(* Logix 5000 project; controller R1USB70001_CWRU_Scenario_Gen_20111116 vendor 1 type 14 code 54 rev 19.11; software revision 19.01; part 5 of 9 *)
(* tags used below, declared in another part *)
   EditScenarioPv : EditScenarioPv;
   ExecutePv : ExecutePv;
   CalcRemainTimeIndex : DINT;
   CalcTotalTimeIndex : DINT;
   CL_LP_B2_SG : ALIAS FOR ACNR_CP_SG_N5:2:O.4;
   EditScenario : EditScenarioPub;
   Execute : ExecutePub;
   HMI : HMIPub;
   IL_LP_B1_SG : ALIAS FOR ACNR_CP_SG_N5:4:O.1;
   IL_LP_B2_SG : ALIAS FOR ACNR_CP_SG_N5:5:O.4;
   IL_LP_ML_SG : ALIAS FOR ACNR_CP_SG_N5:4:O.0;
   Scenario : Scenario_Def[100];
   TimeTblStepNmbr : DINT;
(* MainProgram, continued *)

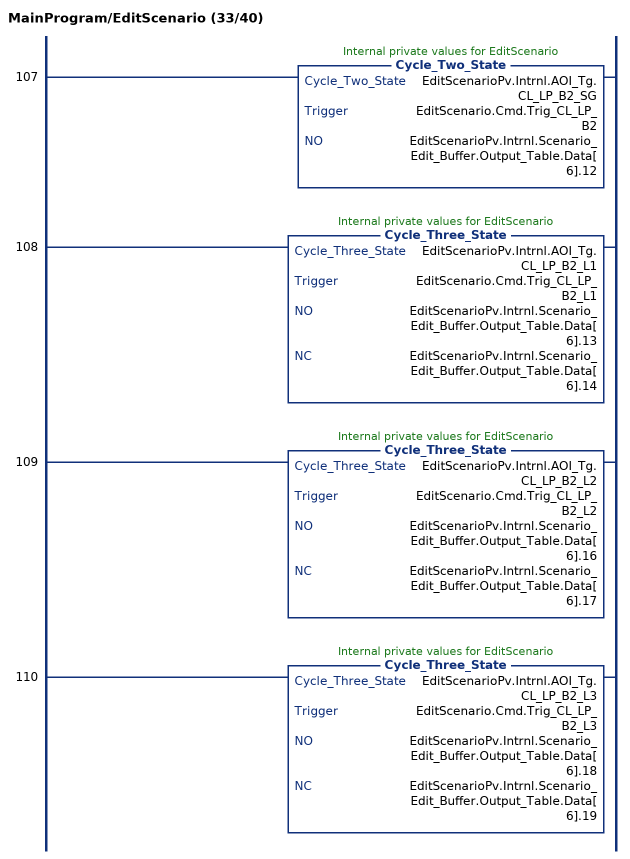
   107: Cycle_Two_State(EditScenarioPv.Intrnl.AOI_Tg.CL_LP_B2_SG,EditScenario.Cmd.Trig_CL_LP_B2,EditScenarioPv.Intrnl.Scenario_Edit_Buffer.Output_Table.Data[6].12);
   108: Cycle_Three_State(EditScenarioPv.Intrnl.AOI_Tg.CL_LP_B2_L1,EditScenario.Cmd.Trig_CL_LP_B2_L1,EditScenarioPv.Intrnl.Scenario_Edit_Buffer.Output_Table.Data[6].13,EditScenarioPv.Intrnl.Scenario_Edit_Buffer.Output_Table.Data[6].14);
   109: Cycle_Three_State(EditScenarioPv.Intrnl.AOI_Tg.CL_LP_B2_L2,EditScenario.Cmd.Trig_CL_LP_B2_L2,EditScenarioPv.Intrnl.Scenario_Edit_Buffer.Output_Table.Data[6].16,EditScenarioPv.Intrnl.Scenario_Edit_Buffer.Output_Table.Data[6].17);
   110: Cycle_Three_State(EditScenarioPv.Intrnl.AOI_Tg.CL_LP_B2_L3,EditScenario.Cmd.Trig_CL_LP_B2_L3,EditScenarioPv.Intrnl.Scenario_Edit_Buffer.Output_Table.Data[6].18,EditScenarioPv.Intrnl.Scenario_Edit_Buffer.Output_Table.Data[6].19);
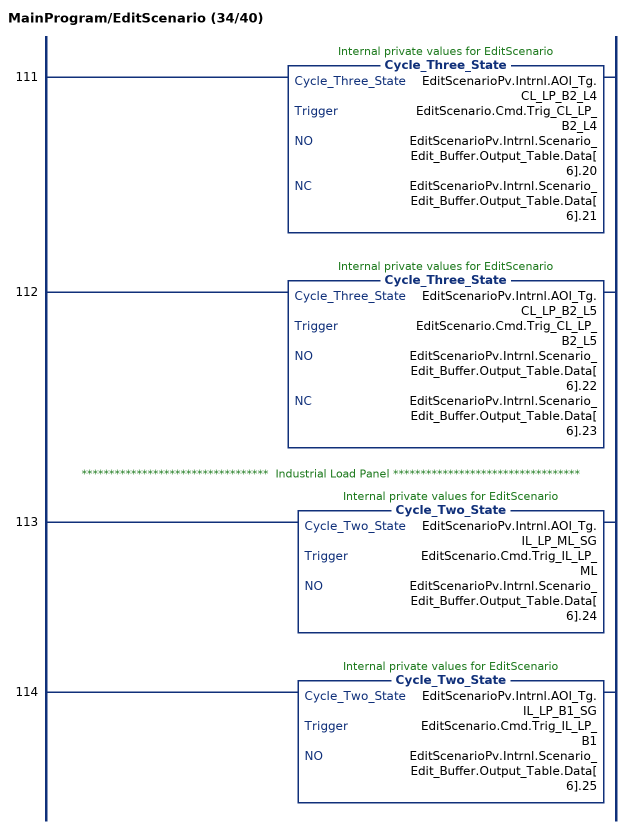
   111: Cycle_Three_State(EditScenarioPv.Intrnl.AOI_Tg.CL_LP_B2_L4,EditScenario.Cmd.Trig_CL_LP_B2_L4,EditScenarioPv.Intrnl.Scenario_Edit_Buffer.Output_Table.Data[6].20,EditScenarioPv.Intrnl.Scenario_Edit_Buffer.Output_Table.Data[6].21);
   112: Cycle_Three_State(EditScenarioPv.Intrnl.AOI_Tg.CL_LP_B2_L5,EditScenario.Cmd.Trig_CL_LP_B2_L5,EditScenarioPv.Intrnl.Scenario_Edit_Buffer.Output_Table.Data[6].22,EditScenarioPv.Intrnl.Scenario_Edit_Buffer.Output_Table.Data[6].23);
   // **********************************  Industrial Load Panel **********************************
   113: Cycle_Two_State(EditScenarioPv.Intrnl.AOI_Tg.IL_LP_ML_SG,EditScenario.Cmd.Trig_IL_LP_ML,EditScenarioPv.Intrnl.Scenario_Edit_Buffer.Output_Table.Data[6].24);
   114: Cycle_Two_State(EditScenarioPv.Intrnl.AOI_Tg.IL_LP_B1_SG,EditScenario.Cmd.Trig_IL_LP_B1,EditScenarioPv.Intrnl.Scenario_Edit_Buffer.Output_Table.Data[6].25);
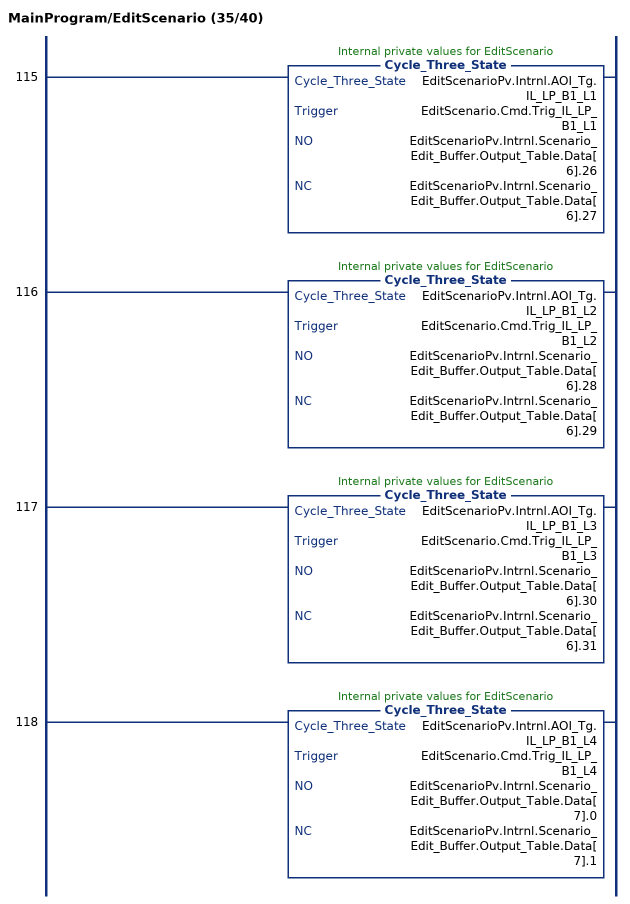
   115: Cycle_Three_State(EditScenarioPv.Intrnl.AOI_Tg.IL_LP_B1_L1,EditScenario.Cmd.Trig_IL_LP_B1_L1,EditScenarioPv.Intrnl.Scenario_Edit_Buffer.Output_Table.Data[6].26,EditScenarioPv.Intrnl.Scenario_Edit_Buffer.Output_Table.Data[6].27);
   116: Cycle_Three_State(EditScenarioPv.Intrnl.AOI_Tg.IL_LP_B1_L2,EditScenario.Cmd.Trig_IL_LP_B1_L2,EditScenarioPv.Intrnl.Scenario_Edit_Buffer.Output_Table.Data[6].28,EditScenarioPv.Intrnl.Scenario_Edit_Buffer.Output_Table.Data[6].29);
   117: Cycle_Three_State(EditScenarioPv.Intrnl.AOI_Tg.IL_LP_B1_L3,EditScenario.Cmd.Trig_IL_LP_B1_L3,EditScenarioPv.Intrnl.Scenario_Edit_Buffer.Output_Table.Data[6].30,EditScenarioPv.Intrnl.Scenario_Edit_Buffer.Output_Table.Data[6].31);
   118: Cycle_Three_State(EditScenarioPv.Intrnl.AOI_Tg.IL_LP_B1_L4,EditScenario.Cmd.Trig_IL_LP_B1_L4,EditScenarioPv.Intrnl.Scenario_Edit_Buffer.Output_Table.Data[7].0,EditScenarioPv.Intrnl.Scenario_Edit_Buffer.Output_Table.Data[7].1);
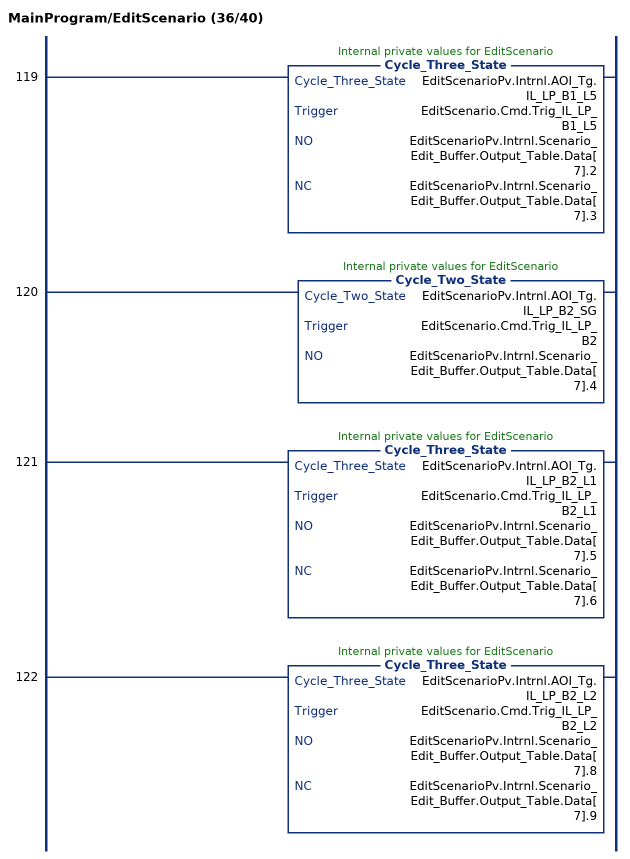
   119: Cycle_Three_State(EditScenarioPv.Intrnl.AOI_Tg.IL_LP_B1_L5,EditScenario.Cmd.Trig_IL_LP_B1_L5,EditScenarioPv.Intrnl.Scenario_Edit_Buffer.Output_Table.Data[7].2,EditScenarioPv.Intrnl.Scenario_Edit_Buffer.Output_Table.Data[7].3);
   120: Cycle_Two_State(EditScenarioPv.Intrnl.AOI_Tg.IL_LP_B2_SG,EditScenario.Cmd.Trig_IL_LP_B2,EditScenarioPv.Intrnl.Scenario_Edit_Buffer.Output_Table.Data[7].4);
   121: Cycle_Three_State(EditScenarioPv.Intrnl.AOI_Tg.IL_LP_B2_L1,EditScenario.Cmd.Trig_IL_LP_B2_L1,EditScenarioPv.Intrnl.Scenario_Edit_Buffer.Output_Table.Data[7].5,EditScenarioPv.Intrnl.Scenario_Edit_Buffer.Output_Table.Data[7].6);
   122: Cycle_Three_State(EditScenarioPv.Intrnl.AOI_Tg.IL_LP_B2_L2,EditScenario.Cmd.Trig_IL_LP_B2_L2,EditScenarioPv.Intrnl.Scenario_Edit_Buffer.Output_Table.Data[7].8,EditScenarioPv.Intrnl.Scenario_Edit_Buffer.Output_Table.Data[7].9);
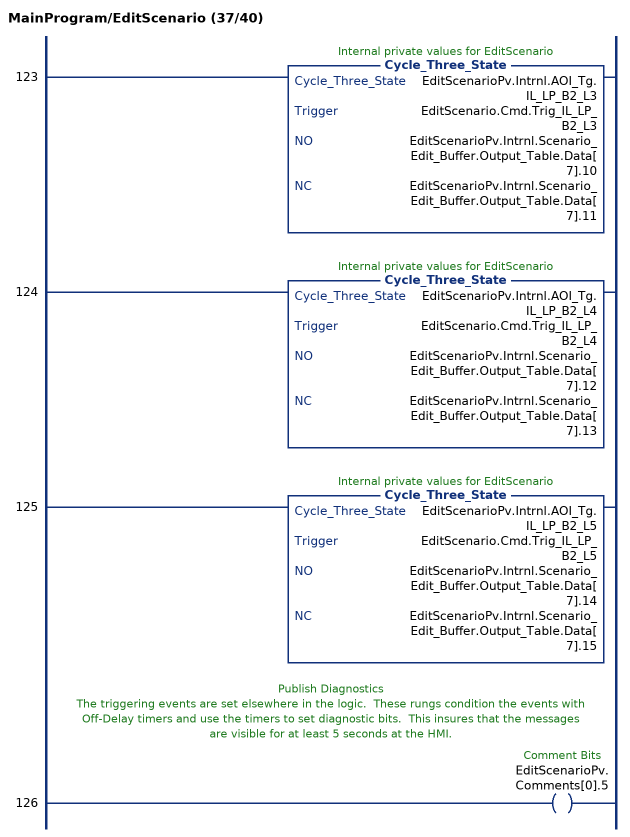
   123: Cycle_Three_State(EditScenarioPv.Intrnl.AOI_Tg.IL_LP_B2_L3,EditScenario.Cmd.Trig_IL_LP_B2_L3,EditScenarioPv.Intrnl.Scenario_Edit_Buffer.Output_Table.Data[7].10,EditScenarioPv.Intrnl.Scenario_Edit_Buffer.Output_Table.Data[7].11);
   124: Cycle_Three_State(EditScenarioPv.Intrnl.AOI_Tg.IL_LP_B2_L4,EditScenario.Cmd.Trig_IL_LP_B2_L4,EditScenarioPv.Intrnl.Scenario_Edit_Buffer.Output_Table.Data[7].12,EditScenarioPv.Intrnl.Scenario_Edit_Buffer.Output_Table.Data[7].13);
   125: Cycle_Three_State(EditScenarioPv.Intrnl.AOI_Tg.IL_LP_B2_L5,EditScenario.Cmd.Trig_IL_LP_B2_L5,EditScenarioPv.Intrnl.Scenario_Edit_Buffer.Output_Table.Data[7].14,EditScenarioPv.Intrnl.Scenario_Edit_Buffer.Output_Table.Data[7].15);
   // Publish Diagnostics
   // The triggering events are set elsewhere in the logic.  These rungs condition the events with Off-Delay timers and use the timers to set diagnostic bits.  This insures that the messages are visible for at least 5 seconds at the HMI.
   126: OTE(EditScenarioPv.Comments[0].5);
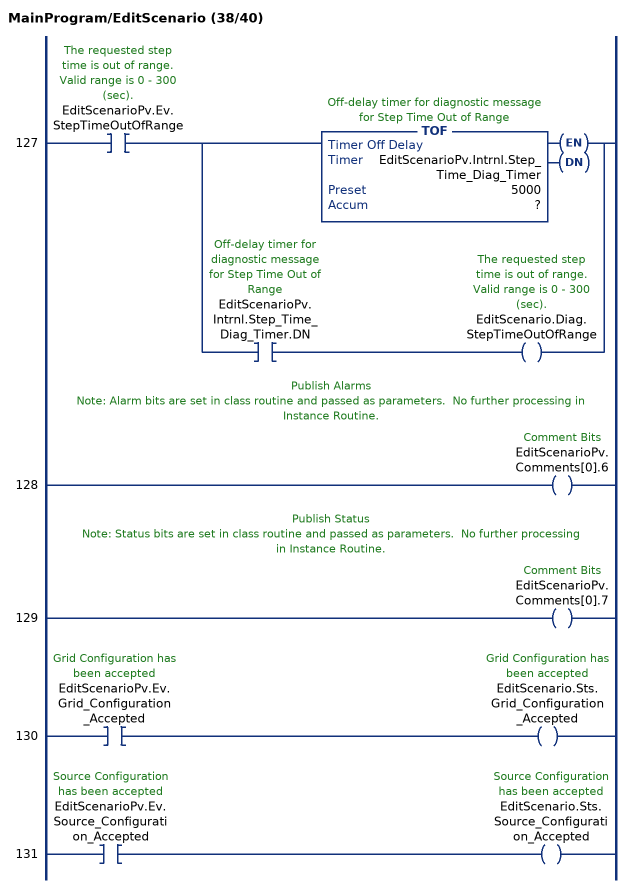
   127: XIC(EditScenarioPv.Ev.StepTimeOutOfRange)[TOF(EditScenarioPv.Intrnl.Step_Time_Diag_Timer,?,?) ,XIC(EditScenarioPv.Intrnl.Step_Time_Diag_Timer.DN) OTE(EditScenario.Diag.StepTimeOutOfRange) ];
   // Publish Alarms
   // Note: Alarm bits are set in class routine and passed as parameters.  No further processing in Instance Routine.
   128: OTE(EditScenarioPv.Comments[0].6);
   // Publish Status
   // Note: Status bits are set in class routine and passed as parameters.  No further processing in Instance Routine.
   129: OTE(EditScenarioPv.Comments[0].7);
   130: XIC(EditScenarioPv.Ev.Grid_Configuration_Accepted)OTE(EditScenario.Sts.Grid_Configuration_Accepted);
   131: XIC(EditScenarioPv.Ev.Source_Configuration_Accepted)OTE(EditScenario.Sts.Source_Configuration_Accepted);
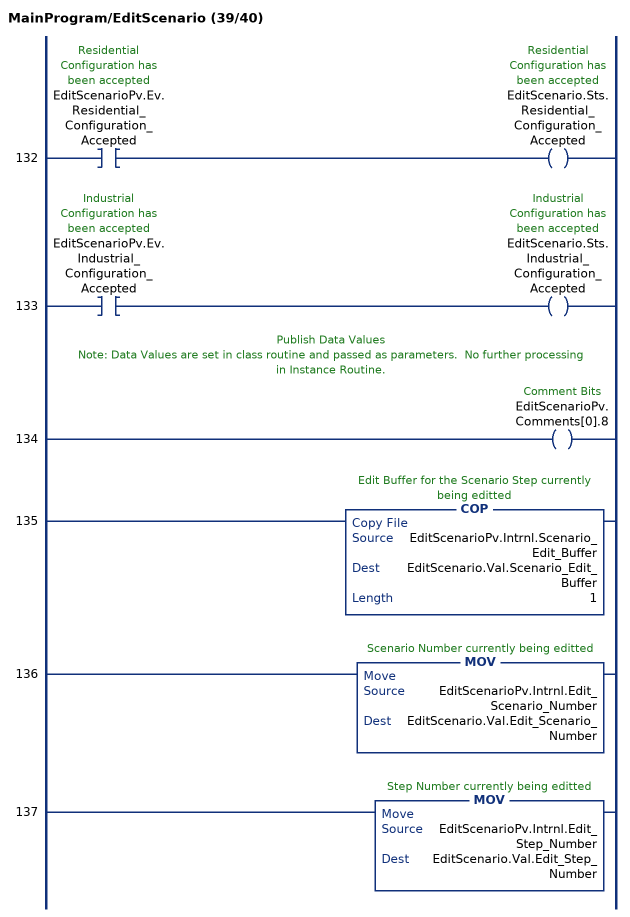
   132: XIC(EditScenarioPv.Ev.Residential_Configuration_Accepted)OTE(EditScenario.Sts.Residential_Configuration_Accepted);
   133: XIC(EditScenarioPv.Ev.Industrial_Configuration_Accepted)OTE(EditScenario.Sts.Industrial_Configuration_Accepted);
   // Publish Data Values
   // Note: Data Values are set in class routine and passed as parameters.  No further processing in Instance Routine.
   134: OTE(EditScenarioPv.Comments[0].8);
   135: COP(EditScenarioPv.Intrnl.Scenario_Edit_Buffer,EditScenario.Val.Scenario_Edit_Buffer,1);
   136: MOV(EditScenarioPv.Intrnl.Edit_Scenario_Number,EditScenario.Val.Edit_Scenario_Number);
   137: MOV(EditScenarioPv.Intrnl.Edit_Step_Number,EditScenario.Val.Edit_Step_Number);
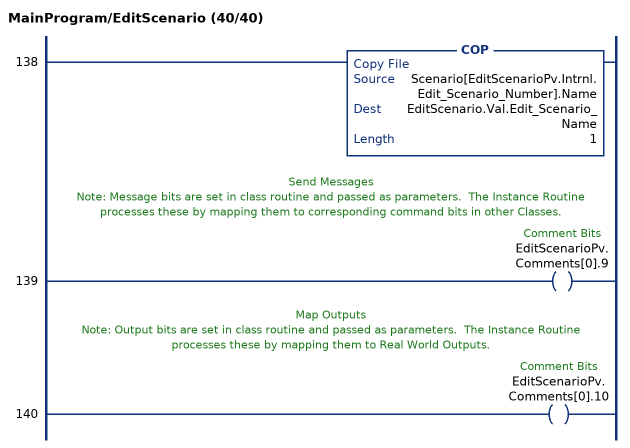
   138: COP(Scenario[EditScenarioPv.Intrnl.Edit_Scenario_Number].Name,EditScenario.Val.Edit_Scenario_Name,1);
   // Send Messages
   // Note: Message bits are set in class routine and passed as parameters.  The Instance Routine processes these by mapping them to corresponding command bits in other Classes.
   139: OTE(EditScenarioPv.Comments[0].9);
   // Map Outputs
   // Note: Output bits are set in class routine and passed as parameters.  The Instance Routine processes these by mapping them to Real World Outputs.
   140: OTE(EditScenarioPv.Comments[0].10);
END_ROUTINE

ROUTINE Execute   (* ladder *)
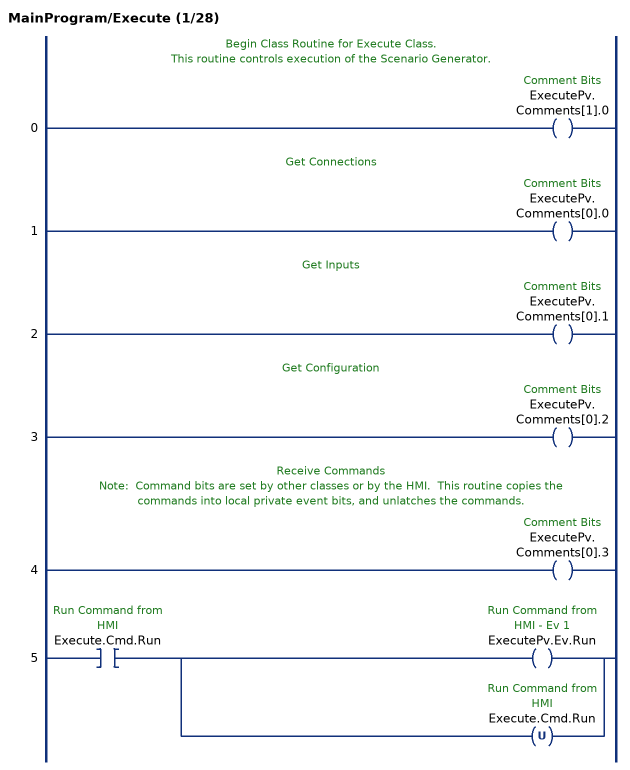
   // Begin Class Routine for Execute Class.
   // This routine controls execution of the Scenario Generator.
   0: OTE(ExecutePv.Comments[1].0);
   // Get Connections
   1: OTE(ExecutePv.Comments[0].0);
   // Get Inputs
   2: OTE(ExecutePv.Comments[0].1);
   // Get Configuration
   3: OTE(ExecutePv.Comments[0].2);
   // Receive Commands
   // Note:  Command bits are set by other classes or by the HMI.  This routine copies the commands into local private event bits, and unlatches the commands.
   4: OTE(ExecutePv.Comments[0].3);
   5: XIC(Execute.Cmd.Run)[OTE(ExecutePv.Ev.Run) ,OTU(Execute.Cmd.Run) ];
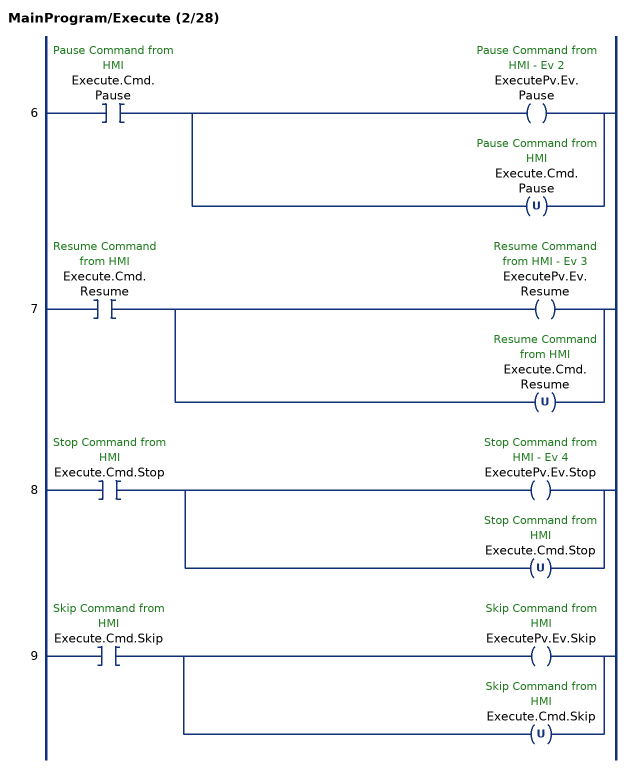
   6: XIC(Execute.Cmd.Pause)[OTE(ExecutePv.Ev.Pause) ,OTU(Execute.Cmd.Pause) ];
   7: XIC(Execute.Cmd.Resume)[OTE(ExecutePv.Ev.Resume) ,OTU(Execute.Cmd.Resume) ];
   8: XIC(Execute.Cmd.Stop)[OTE(ExecutePv.Ev.Stop) ,OTU(Execute.Cmd.Stop) ];
   9: XIC(Execute.Cmd.Skip)[OTE(ExecutePv.Ev.Skip) ,OTU(Execute.Cmd.Skip) ];
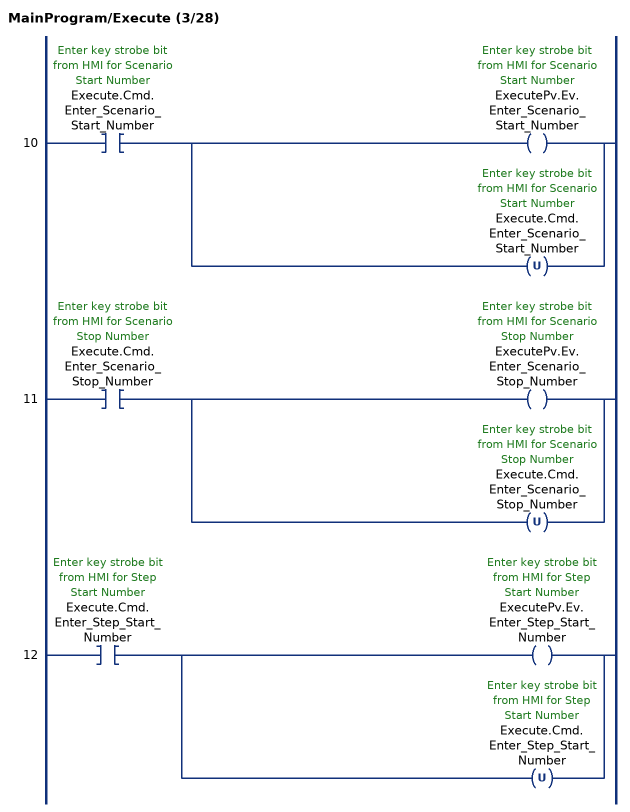
   10: XIC(Execute.Cmd.Enter_Scenario_Start_Number)[OTE(ExecutePv.Ev.Enter_Scenario_Start_Number) ,OTU(Execute.Cmd.Enter_Scenario_Start_Number) ];
   11: XIC(Execute.Cmd.Enter_Scenario_Stop_Number)[OTE(ExecutePv.Ev.Enter_Scenario_Stop_Number) ,OTU(Execute.Cmd.Enter_Scenario_Stop_Number) ];
   12: XIC(Execute.Cmd.Enter_Step_Start_Number)[OTE(ExecutePv.Ev.Enter_Step_Start_Number) ,OTU(Execute.Cmd.Enter_Step_Start_Number) ];
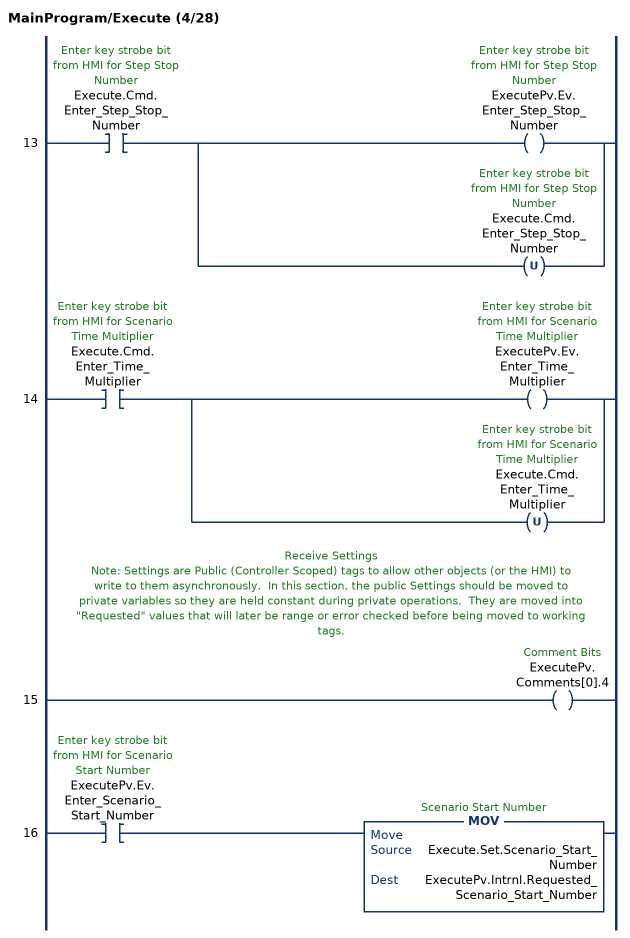
   13: XIC(Execute.Cmd.Enter_Step_Stop_Number)[OTE(ExecutePv.Ev.Enter_Step_Stop_Number) ,OTU(Execute.Cmd.Enter_Step_Stop_Number) ];
   14: XIC(Execute.Cmd.Enter_Time_Multiplier)[OTE(ExecutePv.Ev.Enter_Time_Multiplier) ,OTU(Execute.Cmd.Enter_Time_Multiplier) ];
   // Receive Settings
   // Note: Settings are Public (Controller Scoped) tags to allow other objects (or the HMI) to write to them asynchronously.  In this section, the public Settings should be moved to private variables so they are held constant during private operations.  They are moved into "Requested" values that will later be range or error checked before being moved to working tags.
   15: OTE(ExecutePv.Comments[0].4);
   16: XIC(ExecutePv.Ev.Enter_Scenario_Start_Number)MOV(Execute.Set.Scenario_Start_Number,ExecutePv.Intrnl.Requested_Scenario_Start_Number);
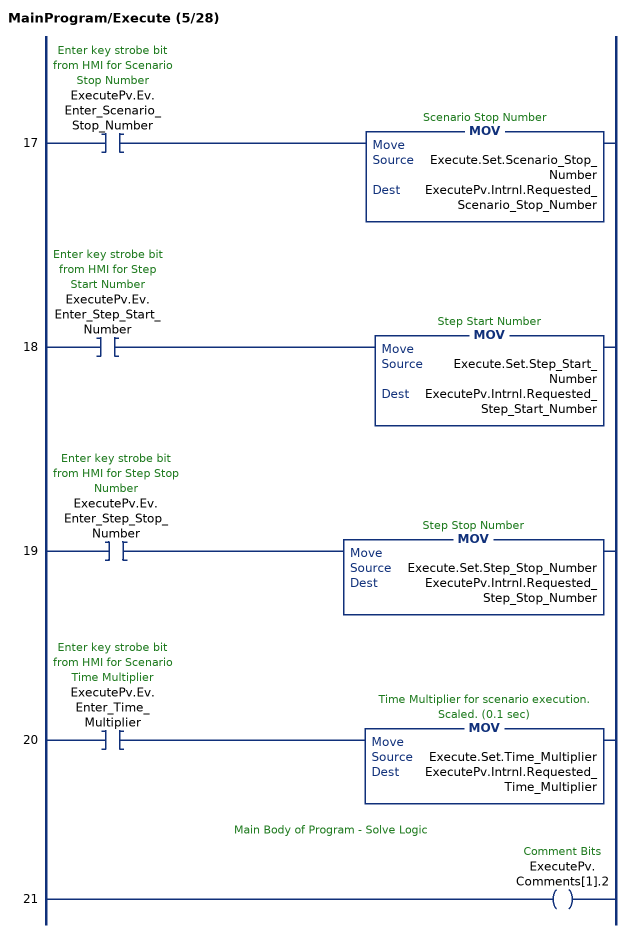
   17: XIC(ExecutePv.Ev.Enter_Scenario_Stop_Number)MOV(Execute.Set.Scenario_Stop_Number,ExecutePv.Intrnl.Requested_Scenario_Stop_Number);
   18: XIC(ExecutePv.Ev.Enter_Step_Start_Number)MOV(Execute.Set.Step_Start_Number,ExecutePv.Intrnl.Requested_Step_Start_Number);
   19: XIC(ExecutePv.Ev.Enter_Step_Stop_Number)MOV(Execute.Set.Step_Stop_Number,ExecutePv.Intrnl.Requested_Step_Stop_Number);
   20: XIC(ExecutePv.Ev.Enter_Time_Multiplier)MOV(Execute.Set.Time_Multiplier,ExecutePv.Intrnl.Requested_Time_Multiplier);
   // Main Body of Program - Solve Logic
   21: OTE(ExecutePv.Comments[1].2);
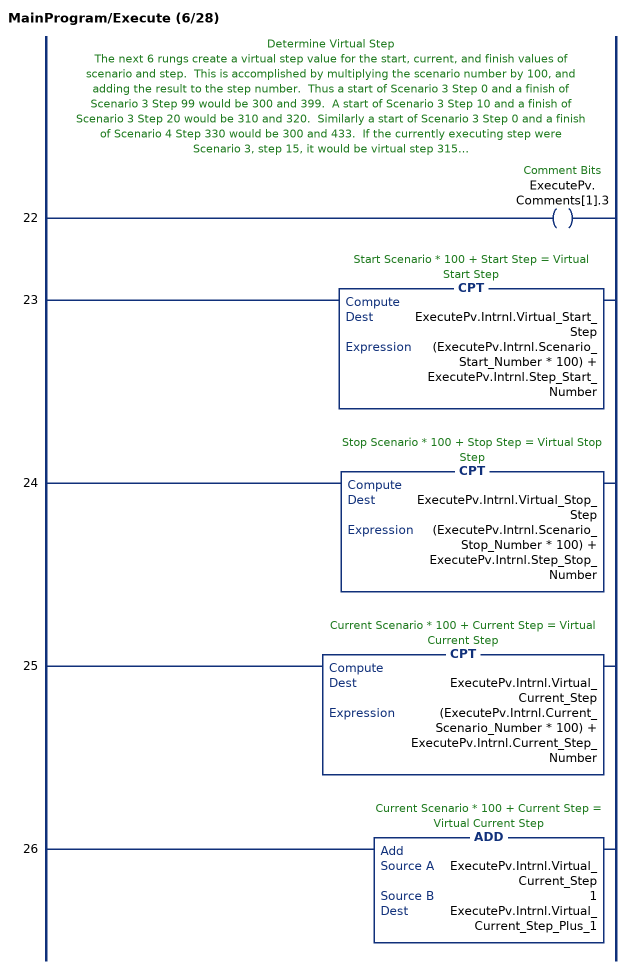
   // Determine Virtual Step
   // The next 6 rungs create a virtual step value for the start, current, and finish values of scenario and step.  This is accomplished by multiplying the scenario number by 100, and adding the result to the step number.  Thus a start of Scenario 3 Step 0 and a finish of Scenario 3 Step 99 would be 300 and 399.  A start of Scenario 3 Step 10 and a finish of Scenario 3 Step 20 would be 310 and 320.  Similarly a start of Scenario 3 Step 0 and a finish of Scenario 4 Step 330 would be 300 and 433.  If the currently executing step were Scenario 3, step 15, it would be virtual step 315.
   // These virtual step values for start, current, and finish will be used to calculate total times and reamining times for scenario execution, and for error checking of start and stop value entries.
   22: OTE(ExecutePv.Comments[1].3);
   23: CPT(ExecutePv.Intrnl.Virtual_Start_Step,(ExecutePv.Intrnl.Scenario_Start_Number * 100) + ExecutePv.Intrnl.Step_Start_Number);
   24: CPT(ExecutePv.Intrnl.Virtual_Stop_Step,(ExecutePv.Intrnl.Scenario_Stop_Number * 100) + ExecutePv.Intrnl.Step_Stop_Number);
   25: CPT(ExecutePv.Intrnl.Virtual_Current_Step,(ExecutePv.Intrnl.Current_Scenario_Number * 100) + ExecutePv.Intrnl.Current_Step_Number);
   26: ADD(ExecutePv.Intrnl.Virtual_Current_Step,1,ExecutePv.Intrnl.Virtual_Current_Step_Plus_1);
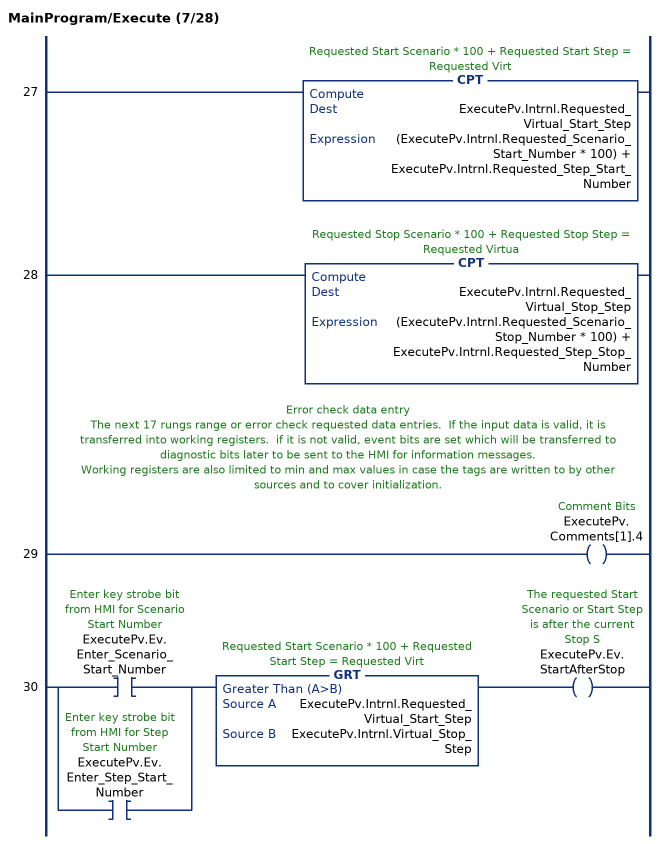
   27: CPT(ExecutePv.Intrnl.Requested_Virtual_Start_Step,(ExecutePv.Intrnl.Requested_Scenario_Start_Number * 100) + ExecutePv.Intrnl.Requested_Step_Start_Number);
   28: CPT(ExecutePv.Intrnl.Requested_Virtual_Stop_Step,(ExecutePv.Intrnl.Requested_Scenario_Stop_Number * 100) + ExecutePv.Intrnl.Requested_Step_Stop_Number);
   // Error check data entry
   // The next 17 rungs range or error check requested data entries.  If the input data is valid, it is transferred into working registers.  if it is not valid, event bits are set which will be transferred to diagnostic bits later to be sent to the HMI for information messages.
   // Working registers are also limited to min and max values in case the tags are written to by other sources and to cover initialization.
   29: OTE(ExecutePv.Comments[1].4);
   30: [XIC(ExecutePv.Ev.Enter_Scenario_Start_Number) ,XIC(ExecutePv.Ev.Enter_Step_Start_Number) ]GRT(ExecutePv.Intrnl.Requested_Virtual_Start_Step,ExecutePv.Intrnl.Virtual_Stop_Step)OTE(ExecutePv.Ev.StartAfterStop);
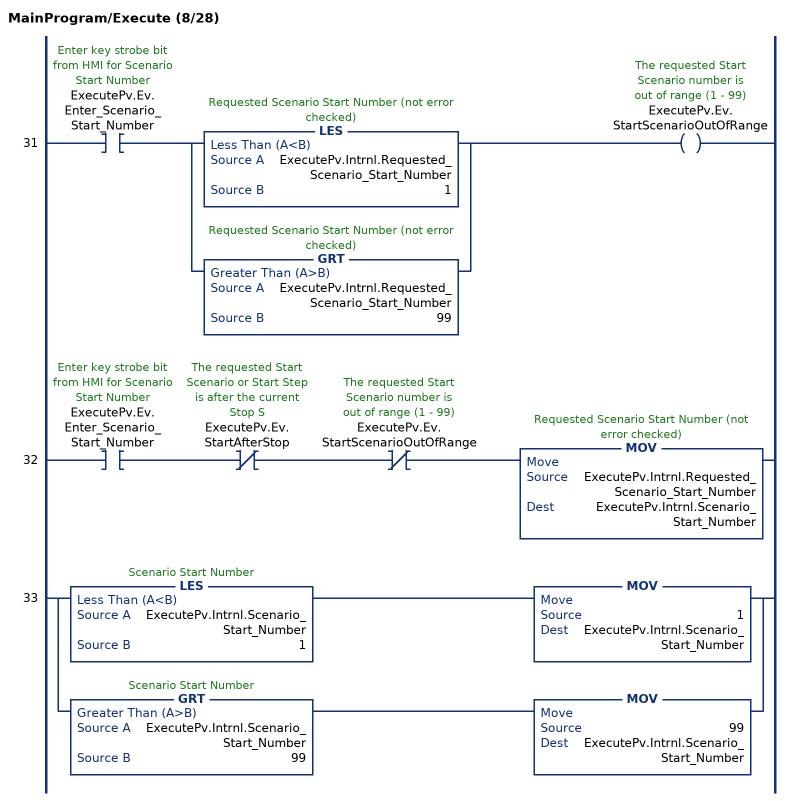
   31: XIC(ExecutePv.Ev.Enter_Scenario_Start_Number)[LES(ExecutePv.Intrnl.Requested_Scenario_Start_Number,1) ,GRT(ExecutePv.Intrnl.Requested_Scenario_Start_Number,99) ]OTE(ExecutePv.Ev.StartScenarioOutOfRange);
   32: XIC(ExecutePv.Ev.Enter_Scenario_Start_Number)XIO(ExecutePv.Ev.StartAfterStop)XIO(ExecutePv.Ev.StartScenarioOutOfRange)MOV(ExecutePv.Intrnl.Requested_Scenario_Start_Number,ExecutePv.Intrnl.Scenario_Start_Number);
   33: [LES(ExecutePv.Intrnl.Scenario_Start_Number,1) MOV(1,ExecutePv.Intrnl.Scenario_Start_Number) ,GRT(ExecutePv.Intrnl.Scenario_Start_Number,99) MOV(99,ExecutePv.Intrnl.Scenario_Start_Number) ];
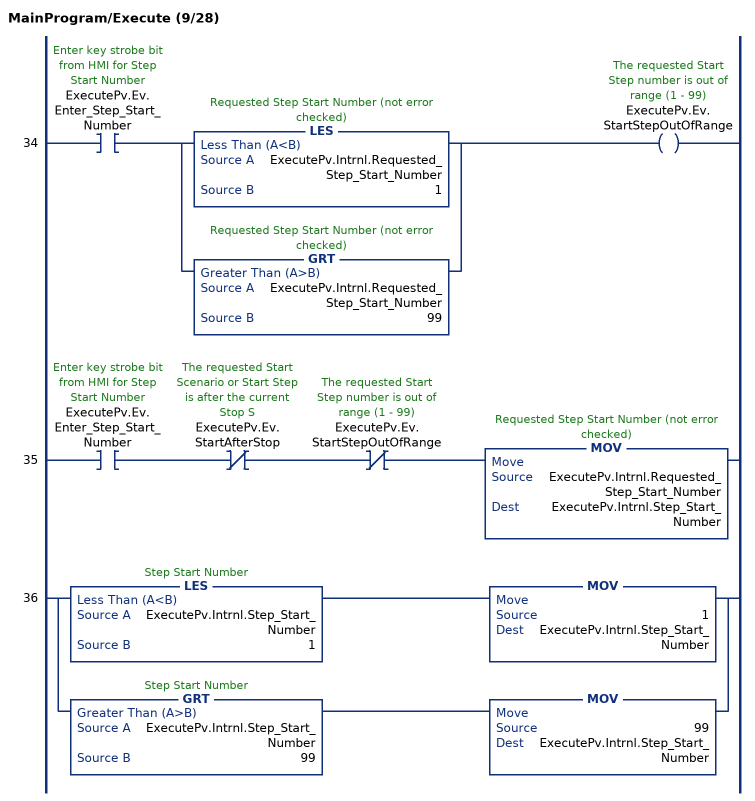
   34: XIC(ExecutePv.Ev.Enter_Step_Start_Number)[LES(ExecutePv.Intrnl.Requested_Step_Start_Number,1) ,GRT(ExecutePv.Intrnl.Requested_Step_Start_Number,99) ]OTE(ExecutePv.Ev.StartStepOutOfRange);
   35: XIC(ExecutePv.Ev.Enter_Step_Start_Number)XIO(ExecutePv.Ev.StartAfterStop)XIO(ExecutePv.Ev.StartStepOutOfRange)MOV(ExecutePv.Intrnl.Requested_Step_Start_Number,ExecutePv.Intrnl.Step_Start_Number);
   36: [LES(ExecutePv.Intrnl.Step_Start_Number,1) MOV(1,ExecutePv.Intrnl.Step_Start_Number) ,GRT(ExecutePv.Intrnl.Step_Start_Number,99) MOV(99,ExecutePv.Intrnl.Step_Start_Number) ];
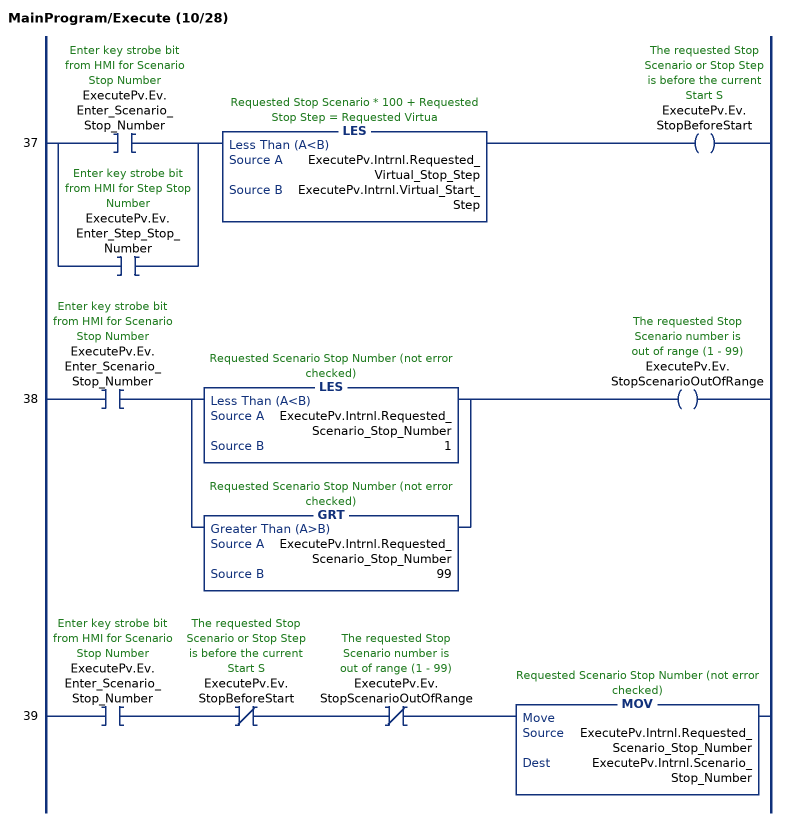
   37: [XIC(ExecutePv.Ev.Enter_Scenario_Stop_Number) ,XIC(ExecutePv.Ev.Enter_Step_Stop_Number) ]LES(ExecutePv.Intrnl.Requested_Virtual_Stop_Step,ExecutePv.Intrnl.Virtual_Start_Step)OTE(ExecutePv.Ev.StopBeforeStart);
   38: XIC(ExecutePv.Ev.Enter_Scenario_Stop_Number)[LES(ExecutePv.Intrnl.Requested_Scenario_Stop_Number,1) ,GRT(ExecutePv.Intrnl.Requested_Scenario_Stop_Number,99) ]OTE(ExecutePv.Ev.StopScenarioOutOfRange);
   39: XIC(ExecutePv.Ev.Enter_Scenario_Stop_Number)XIO(ExecutePv.Ev.StopBeforeStart)XIO(ExecutePv.Ev.StopScenarioOutOfRange)MOV(ExecutePv.Intrnl.Requested_Scenario_Stop_Number,ExecutePv.Intrnl.Scenario_Stop_Number);
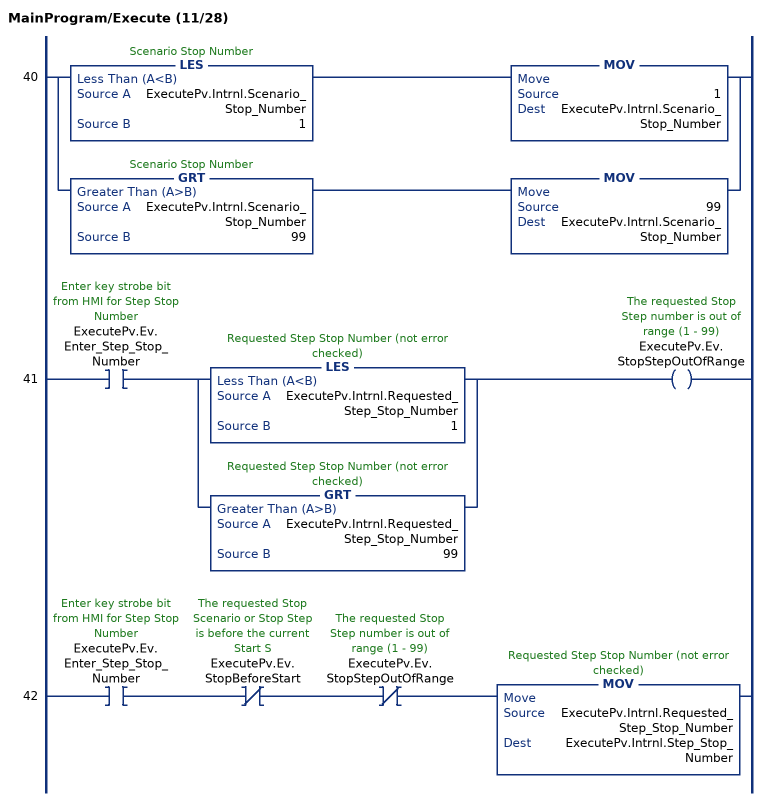
   40: [LES(ExecutePv.Intrnl.Scenario_Stop_Number,1) MOV(1,ExecutePv.Intrnl.Scenario_Stop_Number) ,GRT(ExecutePv.Intrnl.Scenario_Stop_Number,99) MOV(99,ExecutePv.Intrnl.Scenario_Stop_Number) ];
   41: XIC(ExecutePv.Ev.Enter_Step_Stop_Number)[LES(ExecutePv.Intrnl.Requested_Step_Stop_Number,1) ,GRT(ExecutePv.Intrnl.Requested_Step_Stop_Number,99) ]OTE(ExecutePv.Ev.StopStepOutOfRange);
   42: XIC(ExecutePv.Ev.Enter_Step_Stop_Number)XIO(ExecutePv.Ev.StopBeforeStart)XIO(ExecutePv.Ev.StopStepOutOfRange)MOV(ExecutePv.Intrnl.Requested_Step_Stop_Number,ExecutePv.Intrnl.Step_Stop_Number);
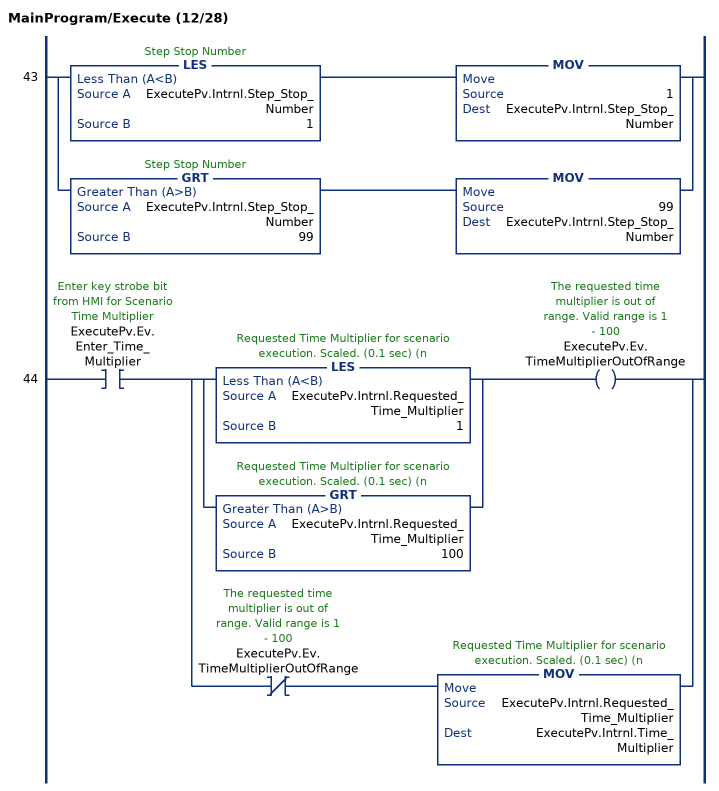
   43: [LES(ExecutePv.Intrnl.Step_Stop_Number,1) MOV(1,ExecutePv.Intrnl.Step_Stop_Number) ,GRT(ExecutePv.Intrnl.Step_Stop_Number,99) MOV(99,ExecutePv.Intrnl.Step_Stop_Number) ];
   44: XIC(ExecutePv.Ev.Enter_Time_Multiplier)[[LES(ExecutePv.Intrnl.Requested_Time_Multiplier,1) ,GRT(ExecutePv.Intrnl.Requested_Time_Multiplier,100) ] OTE(ExecutePv.Ev.TimeMultiplierOutOfRange) ,XIO(ExecutePv.Ev.TimeMultiplierOutOfRange) MOV(ExecutePv.Intrnl.Requested_Time_Multiplier,ExecutePv.Intrnl.Time_Multiplier) ];
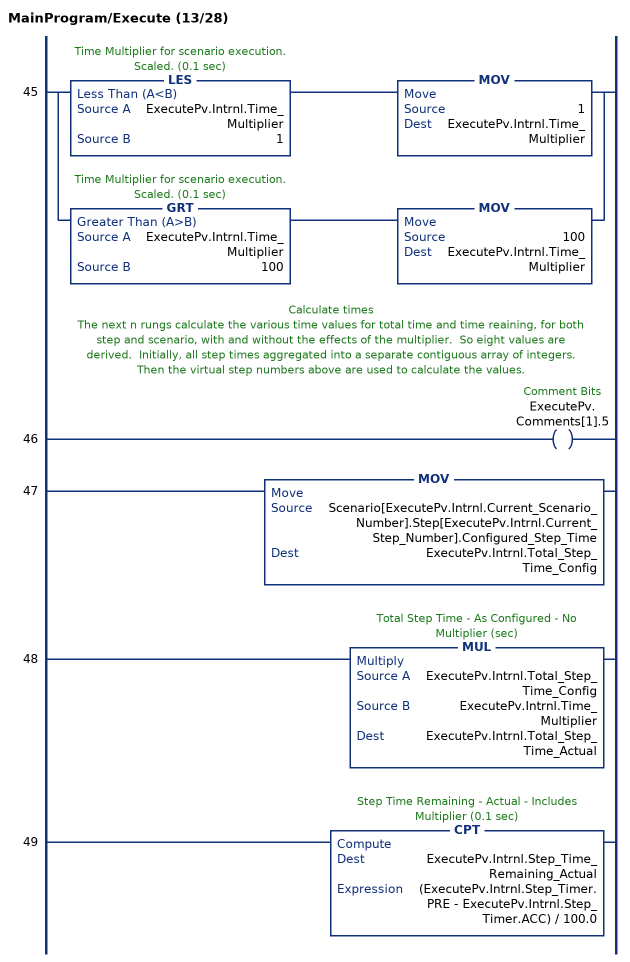
   45: [LES(ExecutePv.Intrnl.Time_Multiplier,1) MOV(1,ExecutePv.Intrnl.Time_Multiplier) ,GRT(ExecutePv.Intrnl.Time_Multiplier,100) MOV(100,ExecutePv.Intrnl.Time_Multiplier) ];
   // Calculate times
   // The next n rungs calculate the various time values for total time and time reaining, for both step and scenario, with and without the effects of the multiplier.  So eight values are derived.  Initially, all step times aggregated into a separate contiguous array of integers.  Then the virtual step numbers above are used to calculate the values.
   46: OTE(ExecutePv.Comments[1].5);
   47: MOV(Scenario[ExecutePv.Intrnl.Current_Scenario_Number].Step[ExecutePv.Intrnl.Current_Step_Number].Configured_Step_Time,ExecutePv.Intrnl.Total_Step_Time_Config);
   48: MUL(ExecutePv.Intrnl.Total_Step_Time_Config,ExecutePv.Intrnl.Time_Multiplier,ExecutePv.Intrnl.Total_Step_Time_Actual);
   49: CPT(ExecutePv.Intrnl.Step_Time_Remaining_Actual,(ExecutePv.Intrnl.Step_Timer.PRE - ExecutePv.Intrnl.Step_Timer.ACC) / 100.0);
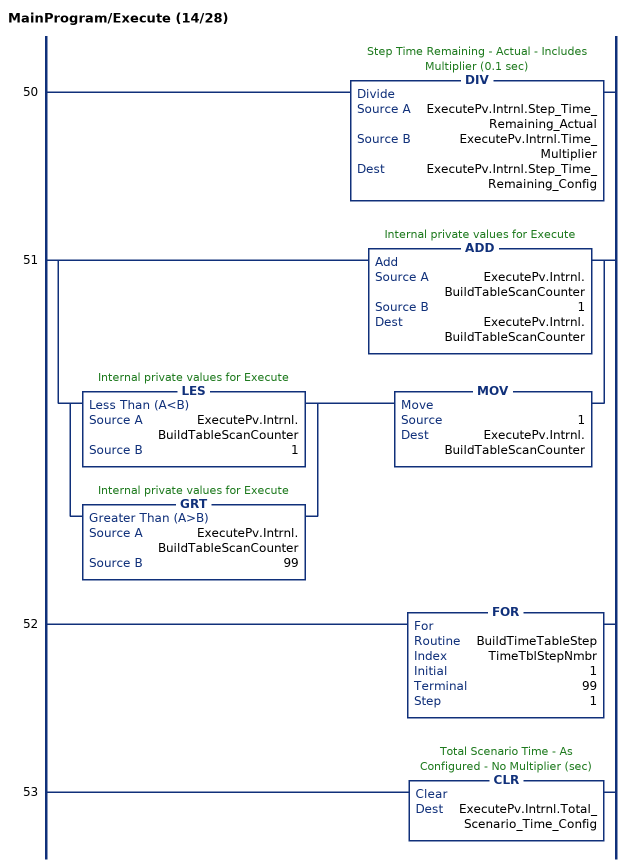
   50: DIV(ExecutePv.Intrnl.Step_Time_Remaining_Actual,ExecutePv.Intrnl.Time_Multiplier,ExecutePv.Intrnl.Step_Time_Remaining_Config);
   51: [ADD(ExecutePv.Intrnl.BuildTableScanCounter,1,ExecutePv.Intrnl.BuildTableScanCounter) ,[LES(ExecutePv.Intrnl.BuildTableScanCounter,1) ,GRT(ExecutePv.Intrnl.BuildTableScanCounter,99) ] MOV(1,ExecutePv.Intrnl.BuildTableScanCounter) ];
   52: FOR(BuildTimeTableStep,TimeTblStepNmbr,1,99,1);
   53: CLR(ExecutePv.Intrnl.Total_Scenario_Time_Config);
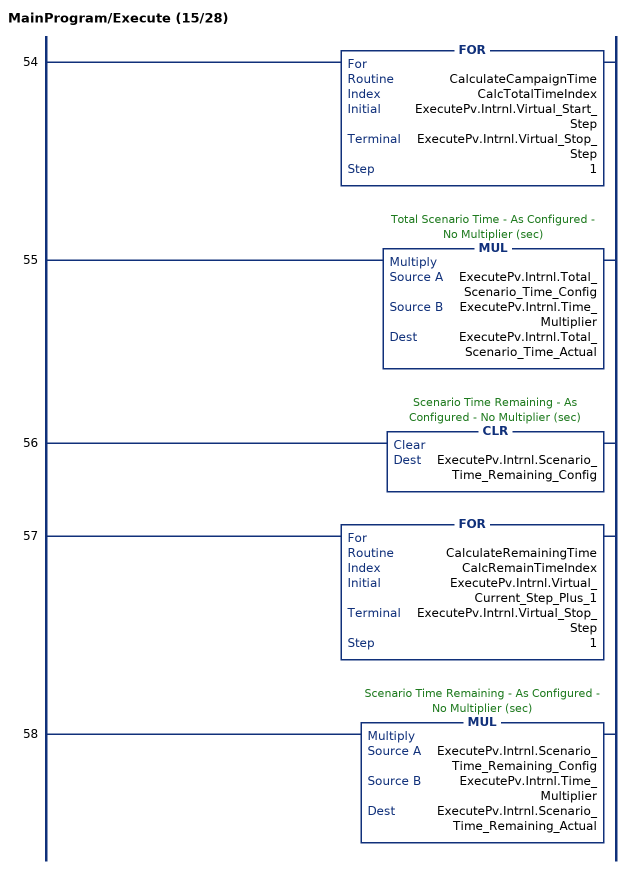
   54: FOR(CalculateCampaignTime,CalcTotalTimeIndex,ExecutePv.Intrnl.Virtual_Start_Step,ExecutePv.Intrnl.Virtual_Stop_Step,1);
   55: MUL(ExecutePv.Intrnl.Total_Scenario_Time_Config,ExecutePv.Intrnl.Time_Multiplier,ExecutePv.Intrnl.Total_Scenario_Time_Actual);
   56: CLR(ExecutePv.Intrnl.Scenario_Time_Remaining_Config);
   57: FOR(CalculateRemainingTime,CalcRemainTimeIndex,ExecutePv.Intrnl.Virtual_Current_Step_Plus_1,ExecutePv.Intrnl.Virtual_Stop_Step,1);
   58: MUL(ExecutePv.Intrnl.Scenario_Time_Remaining_Config,ExecutePv.Intrnl.Time_Multiplier,ExecutePv.Intrnl.Scenario_Time_Remaining_Actual);
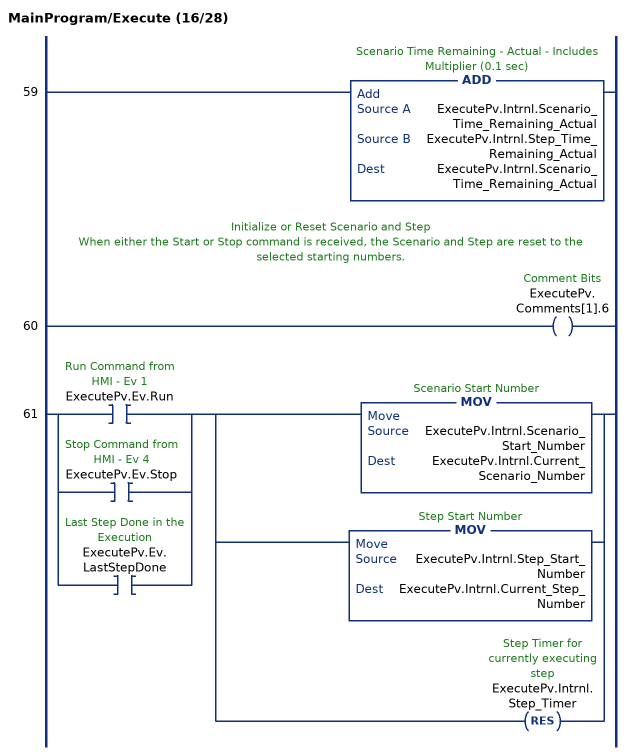
   59: ADD(ExecutePv.Intrnl.Scenario_Time_Remaining_Actual,ExecutePv.Intrnl.Step_Time_Remaining_Actual,ExecutePv.Intrnl.Scenario_Time_Remaining_Actual);
   // Initialize or Reset Scenario and Step
   // When either the Start or Stop command is received, the Scenario and Step are reset to the selected starting numbers.
   60: OTE(ExecutePv.Comments[1].6);
   61: [XIC(ExecutePv.Ev.Run) ,XIC(ExecutePv.Ev.Stop) ,XIC(ExecutePv.Ev.LastStepDone) ][MOV(ExecutePv.Intrnl.Scenario_Start_Number,ExecutePv.Intrnl.Current_Scenario_Number) ,MOV(ExecutePv.Intrnl.Step_Start_Number,ExecutePv.Intrnl.Current_Step_Number) ,RES(ExecutePv.Intrnl.Step_Timer) ];
